DATA_BLOCK "ST10_Flow4_B1Press_iDB"
{ S7_Optimized_Access := 'TRUE' }
VERSION : 0.1
NON_RETAIN
"ST10_Flow4_B1Press"

BEGIN

END_DATA_BLOCK

